Staubli VAL3: home.pjx

--- home.pjx ---
Parameters version=s7.2.1 stackSize=5000 millimeterUnit=true
Data file=home.dtx
Library alias=io path=Disk://io/io.pjx

--- home.dtx ---
public num distance
public num moveType
public num nIndexGun
public num nStop
public num nTcpAction
public num nTime
public string comment
public string instruction
public string sProgram
public bool toStop
public jointRx jJoints
public mdesc nom_speed = {vel=10, tmax=9999, rmax=9999, leave=30, reach=30}
